// LS Electric XG5000 project: 8_23_2
// PLC LSPLC

PROGRAM NewProgram (task: 스캔 프로그램)

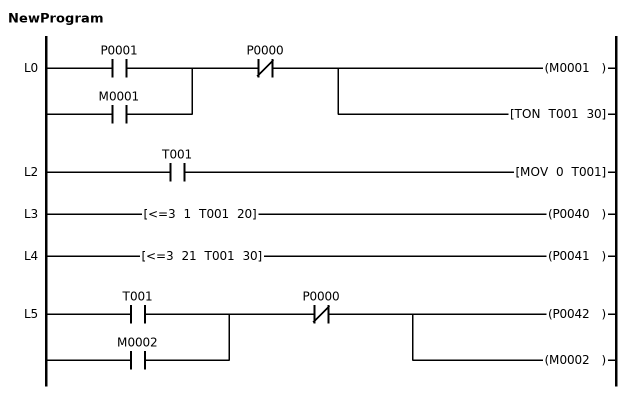
; L0
LOAD      P0001
OR        M0001
AND NOT   P0000
OUT       M0001
TON       T001 30
; L2
LOAD      T001
MOV       0 T001
; L3
LOAD<=3   1 T001 20
OUT       P0040
; L4
LOAD<=3   21 T001 30
OUT       P0041
; L5
LOAD      T001
OR        M0002
AND NOT   P0000
OUT       P0042
OUT       M0002